(* IEC 61131-3 sources: volt/packages/volt-lsp-iec/test-corpus/awa-palletizer/Device/Plc Logic/Application/Library Manager/L_Util, 15 files *)

(* ---- TRETAINERRORID.dut ---- *)
TYPE TRETAINERRORID :
(
	NO_ERROR := 0,
	RETAIN_DATA_NOT_STORED := 1,
	MORE_THAN_ONE_INSTANCE := 2
);
END_TYPE

(* ---- TTARGETIDS.dut ---- *)
TYPE TTARGETIDS :
(
	C3200_LOGIC := 16#100,
	C3241_LOGIC := 16#110,
	P500_LOGIC := 16#180,
	C300_LOGIC := 16#200,
	P300_MOTION := 16#220,
	P300_LOGIC := 16#280
);
END_TYPE

(* ---- TWATCHDOGTIME.dut ---- *)
TYPE TWATCHDOGTIME :
STRUCT
	WDTIMEORIGINAL : DWORD;
	WDTIMECHECK : DWORD;
	IDTASK : UDINT;
	HTASK : RTS_IEC_HANDLE;
END_STRUCT
END_TYPE

(* ---- CALLBACKDELETERETAINFILE.pou ---- *)
FUNCTION CALLBACKDELETERETAINFILE : BOOL
VAR_INPUT
	DWSPEC : DWORD;
	DWPARAM : DWORD;
	DWSOURCE : DWORD;
END_VAR
END_FUNCTION

(* ---- GETBOOLEANPROPERTY.pou ---- *)
FUNCTION GETBOOLEANPROPERTY : BOOL
VAR_INPUT
	STKEY : WSTRING;
END_VAR
END_FUNCTION

(* ---- GETCOMPANY.pou ---- *)
FUNCTION GETCOMPANY : WSTRING
END_FUNCTION

(* ---- GETNUMBERPROPERTY.pou ---- *)
FUNCTION GETNUMBERPROPERTY : DINT
VAR_INPUT
	STKEY : WSTRING;
END_VAR
END_FUNCTION

(* ---- GETTEXTPROPERTY.pou ---- *)
FUNCTION GETTEXTPROPERTY : WSTRING
VAR_INPUT
	STKEY : WSTRING;
END_VAR
END_FUNCTION

(* ---- GETTEXTPROPERTY2.pou ---- *)
FUNCTION GETTEXTPROPERTY2 : POINTER TO WSTRING
VAR_INPUT
	STKEY : WSTRING;
END_VAR
END_FUNCTION

(* ---- GETTITLE.pou ---- *)
FUNCTION GETTITLE : WSTRING
END_FUNCTION

(* ---- GETVERSION.pou ---- *)
FUNCTION GETVERSION : VERSION
END_FUNCTION

(* ---- GETVERSIONPROPERTY.pou ---- *)
FUNCTION GETVERSIONPROPERTY : VERSION
VAR_INPUT
	STKEY : WSTRING;
END_VAR
END_FUNCTION

(* ---- L_SUSPENDWATCHDOG.pou ---- *)
FUNCTION_BLOCK L_SUSPENDWATCHDOG
VAR_INPUT
	BEXECUTE : BOOL := TRUE;
	WNUMBEROFCYCLES : WORD := 20;
END_VAR
VAR
	DICOUNTER : DINT;
	XBUSY : BOOL;
	XBUSYOLD : BOOL;
	BEXECUTEOLD : BOOL;
	BSWITCHCE : BOOL;
	XWAITPLCSTART : BOOL;
	PAPPLICATION : POINTER TO CmpApp.APPLICATION;
	PAPPNAME : POINTER TO STRING(MAX_LEN_APPLNAME);
	PIECTASKRESULT : POINTER TO RTS_IEC_RESULT;
	TIECTASKHANDLE : RTS_IEC_HANDLE;
	PIECTASKINFO : POINTER TO Task_Info2;
	WTASKCOUNT : WORD;
	WTASKCOUNTEVT : WORD;
	RESULT : RTS_IEC_RESULT;
	ERRORCOUNT : WORD;
	XWATCHDOGDISABLED : BOOL;
	DWCALL : DWORD;
	XFIRSTPREPARESTARTEVENTDONE : BOOL;
	ITFCALLBACK : CmpEventMgr.ICmpEventCallback;
	HEVENTPREPARESTART : RTS_IEC_HANDLE := SysTypes.RTS_INVALID_HANDLE;
	HINTERFACEPREPARESTART : RTS_IEC_HANDLE := SysTypes.RTS_INVALID_HANDLE;
	DWEVTCOUNT_PREPAREAPPSTART : DWORD := 0;
END_VAR
END_FUNCTION_BLOCK

METHOD CYCLICCALLINTERN
END_METHOD

METHOD CYCLICCALLINTERN_1
END_METHOD

METHOD EVENTCALLBACK : UDINT
VAR_INPUT
	PEVENTPARAM : POINTER TO EventParam;
END_VAR
END_METHOD

METHOD REGISTEREVENT
END_METHOD

METHOD UNREGISTEREVENT
END_METHOD

METHOD FB_INIT : BOOL
VAR_INPUT
	BINITRETAINS : BOOL;
	BINCOPYCODE : BOOL;
END_VAR
END_METHOD

METHOD FB_EXIT : BOOL
VAR_INPUT
	BINCOPYCODE : BOOL;
END_VAR
END_METHOD

(* ---- L_SUSPENDWATCHDOGSENSITIVE.pou ---- *)
FUNCTION_BLOCK L_SUSPENDWATCHDOGSENSITIVE
VAR_INPUT
	BEXECUTE : BOOL := TRUE;
	WNUMBEROFCYCLES : WORD := 20;
END_VAR
VAR_OUTPUT
	XBUSY : BOOL;
	XWATCHDOGACTIVE : BOOL;
END_VAR
VAR
	CONST_UIWATCHDOGTIMESLENGH : UINT := 16;
	CONST_UIWATCHDOGTIMES_FACTOR : UINT := 3;
	M_XINITDONE : BOOL;
	M_BEXECUTEOLD : BOOL;
	M_DICOUNTDOWN : DINT;
	M_XWAITPLCSTART : BOOL;
	M_XWDDISABLEDBYPREPARESTART : BOOL;
	M_XFIRSTPREPARESTARTEVENTDONE : BOOL;
	M_ITFCALLBACK : CmpEventMgr.ICmpEventCallback;
	M_HEVENTPREPARESTART : RTS_IEC_HANDLE := SysTypes.RTS_INVALID_HANDLE;
	M_HINTERFACEPREPARESTART : RTS_IEC_HANDLE := SysTypes.RTS_INVALID_HANDLE;
	M_PMASTER : POINTER TO L_IODrvEtherCAT;
	M_ISMASTERSYSTEM : BOOL;
	M_WDDISABLEBYMASTER : BOOL;
	M_WDWATCHDOGRAISED : BOOL;
	AWATCHDOGTIMES : ARRAY [0..(CONST_UIWATCHDOGTIMESLENGH - 1)] OF tWatchdogTime;
	M_PTASKS : ARRAY [0..15] OF RTS_IEC_HANDLE;
	M_UINUMOFTASKS : UINT := 0;
	UDIERRCOUNTER : UDINT;
	XDISABLEALLTHISCYCLE : BOOL;
END_VAR
END_FUNCTION_BLOCK

METHOD CYCLICCALLINTERN
END_METHOD

METHOD INITTASKSTRUCT
END_METHOD

METHOD ISECMASTERSYSTEM : BOOL
VAR_INPUT
	UICOM : UINT;
END_VAR
END_METHOD

METHOD ISIECRUNNING : BOOL
END_METHOD

METHOD TRACE : BOOL
VAR_INPUT
	MSG : STRING;
END_VAR
END_METHOD

METHOD WDDISABLEALLTHISCYCLE : DWORD
END_METHOD

METHOD WDENABLEALL : DWORD
END_METHOD

METHOD WDWATCHDOGRAISE : DWORD
END_METHOD

METHOD WDWATCHDOGRESET : DWORD
END_METHOD

METHOD EVENTCALLBACK : UDINT
VAR_INPUT
	PEVENTPARAM : POINTER TO EventParam;
END_VAR
END_METHOD

METHOD REGISTEREVENT
END_METHOD

METHOD UNREGISTEREVENT
END_METHOD

METHOD FB_AFTERGLOABALINIT : BOOL
END_METHOD

METHOD FB_EXIT : BOOL
VAR_INPUT
	BINCOPYCODE : BOOL;
END_VAR
END_METHOD

METHOD FB_INIT : BOOL
VAR_INPUT
	BINITRETAINS : BOOL;
	BINCOPYCODE : BOOL;
END_VAR
END_METHOD

(* ---- L_UTIL_RETAIN.pou ---- *)
FUNCTION_BLOCK L_UTIL_RETAIN
VAR_INPUT
	XSTORERETAINS : BOOL;
END_VAR
VAR_OUTPUT
	XRETAINSSTOREDINTOFILE : BOOL;
	XRETAINSRESTOREDFROMFILE : BOOL;
	XRETAINSRESTOREDFROMMEMORY : BOOL;
	XDONE : BOOL;
	XBUSY : BOOL;
	XERROR : BOOL;
	EERRORID : tRetainErrorId := NO_ERROR;
END_VAR
VAR
	PAPP : POINTER TO APPLICATION;
	PRESULT : POINTER TO RTS_IEC_RESULT;
	STRRETFILE : STRING := 'retains.ret';
	DWTHISINSTANCE : DWORD;
	XSTORERETAINSOLD : BOOL := FALSE;
	MYCALLBACK : CB.CALLBACK;
	PEERROR : POINTER TO CB.ERROR;
	BRESTOREDRETAINDATA : BOOL;
	BRESTOREDMOTIONDATA : BOOL;
	BSTOREDRETAINDATA : BOOL;
	BSTOREDMOTIONDATA : BOOL;
	DWTESTRETAIN : DWORD;
	DWNUMBEROFINSTANCES : DWORD;
END_VAR
END_FUNCTION_BLOCK

METHOD FB_AFTERGLOBALINIT : BOOL
END_METHOD
